Fanuc KAREL source: compact_preamble.KL

PROGRAM KX00001
%NOLOCKGROUP
VAR
I:INTEGER;J:INTEGER;B:BOOLEAN
F : FILE
S : STRING[80]
P : XYZWPR
BEGIN
OPEN FILE F ('RW','MD:KFSAMPLE.DT')
END KX00001
